PROGRAM NasmythControl
VAR_INPUT
	// unlocks the brake and enables the drive
	enable:	BOOL;
	// resets the drive
	reset: BOOL;
	// turns the Nasmyth mirror to left port (seen from top)
	left:	BOOL;
	// turns the Nasmyth mirror to right port (seen from top)
	right:	BOOL;
END_VAR
VAR_OUTPUT
	// Nasmyth drive error
	error:	BOOL;
	// drive ready
	Ready:	BOOL;
END_VAR
VAR
	// axis function block
	Nasmyth_control:	FB_Cover;
	// delay for the Nasmyth holding brake
	Nasmyth_delay:		TON;
	// status word for MQTT message
	Nasmyth_status:		WORD;
	// last status word to trigger MQTT message if different
	LastStatus:			WORD;
	// unlock the holding brake
	Nasmyth_unlock:		BOOL;
	// holding brake is unlocked
	Nasmyth_unlocked:	BOOL;
	// Nasmyth points to right mirror
	Nasmyth_right:		BOOL;
	// Nasmyth points to left mirror
	Nasmyth_left:		BOOL;
	// event log of error
	NasmythEvent: 		FB_Eventlog;
	NasmythLeftEvent:	FB_Eventlog;
	NasmythRightEvent:	FB_Eventlog;
	Nasmyth_Timeout:	TON := (PT := T#10S);
	//MQTTTimer: 			TON := (PT:=T#10S);
	// MQTT String
	sPayloadPub: STRING(255);
END_VAR

// get the inputs
Nasmyth_left := GVL_Telescope.nasmyth_limit_right;
Nasmyth_right := GVL_Telescope.nasmyth_limit_left;

// disable command, if position has been reached or 
IF Nasmyth_left OR right THEN
	left := FALSE;
END_IF

IF  Nasmyth_right OR left THEN
	right := FALSE;
END_IF

Nasmyth_status.0 := Nasmyth_unlocked;
Nasmyth_status.1 := error;
Nasmyth_status.2 := Nasmyth_left;
Nasmyth_status.3 := Nasmyth_right;
Nasmyth_status.4 := Nasmyth_Timeout.Q;

Nasmyth_unlock := enable AND (left OR right);
// report Nasmyth unlocked after n milliseconds										
Nasmyth_delay(
	IN := Nasmyth_unlock,
	PT := T#250MS,
	Q => Nasmyth_unlocked);

// set the outputs
GVL_Telescope.nasmyth_lock := Nasmyth_unlock;
	
Nasmyth_control(
	open := left,
	close := right,
	enable := Nasmyth_unlocked,
	reset := reset,
	limit_open := NOT Nasmyth_left,
	limit_close := NOT Nasmyth_right,
	error => error,
	Ready => ready);

Nasmyth_Timeout(IN := (left AND NOT Nasmyth_left) OR (right AND NOT Nasmyth_right));

IF Nasmyth_status <> LastStatus THEN
	LastStatus := Nasmyth_status;
	sPayloadPub := 'telescope,location=dome,host=CX-22747A,module=NasmythControl ';
	sPayloadPub := APPEND(sPayloadPub, 'NasmythUnlocked=', BOOL_TO_STRING(Nasmyth_unlocked));
	sPayloadPub := APPEND(sPayloadPub, ',NasmythAxisOK=', BOOL_TO_STRING(NOT error));
	sPayloadPub := APPEND(sPayloadPub, ',NasmythIsLeft=', BOOL_TO_STRING(Nasmyth_left));
	sPayloadPub := APPEND(sPayloadPub, ',NasmythIsRight=', BOOL_TO_STRING(Nasmyth_right));
	
	
	MQTTCommunication.fbMqttClient.Publish(	
					sTopic:= 'STELLA1/Telemetry', 
					pPayload:= ADR(sPayloadPub), 
					nPayloadSize:= LEN2(ADR(sPayloadPub)),
					eQoS:= TcIotMqttQos.AtMostOnceDelivery,
					bRetain:= TRUE, 
					bQueue:= FALSE );
END_IF


NasmythEvent(	Trigger := error, 
				Level := ADSLOG_MSGTYPE_ERROR,
				OnMessage := 'Nasmyth axis error',
				OffMessage := 'OK',
				OffLevel := ADSLOG_MSGTYPE_HINT);

NasmythLeftEvent(	Trigger := Nasmyth_left, 
					Level := ADSLOG_MSGTYPE_HINT,
					OnMessage := 'Nasmyth is on left port');

NasmythRightEvent(	Trigger := Nasmyth_right, 
					Level := ADSLOG_MSGTYPE_HINT,
					OnMessage := 'Nasmyth is on right port');

END_PROGRAM

(* stored: Version 1.1.0.1, ProductVersion 3.1.4024.9
   POU NasmythControl: Id {44cc95a4-2714-4f68-86b9-267e29c12088}, SpecialFunc None *)
